// TIA Portal V19 export
FUNCTION_BLOCK "Motor"   // FB126, LAD
TITLE = MOTOR MANAGER / SIMPLE MOTOR MANAGER
// stored: Access Published, MemoryReserve 100, SetENOAutomatically false
   VAR_INPUT
      MotorCtrl : "MotorCtrl";
      ThermalProtection : Bool;   // Thermal protection (0 =OK)
      FdbkRunning : Bool;   // Contactor feedback
      FeedbackTimeout : Time := T#1S;   // Contatr feedback timeout
      Simulation : Bool;   // Simulation device
   END_VAR
   VAR_OUTPUT
      MotorSts : "MotorSts";
      Contactor : Bool;
   END_VAR
   VAR_IN_OUT
      Alarm : "MotorAlr";
   END_VAR
   VAR
      DelayContactorFeedbackON : IEC_TIMER;
      Ctrl_RunContactor : Bool;
   END_VAR
   VAR_TEMP
      DelayOnStart : Bool;
      DelayOffStart : Bool;
      AlarmPresence : Bool;
      RunPermitted : Bool;
   END_VAR
BEGIN

REGION Network 1 (SCL): Info
   //=============================================================================
   //PM FORMING
   //-----------------------------------------------------------------------------
   // Library: StandardBlocks
   // Tested with: S7-1518TF
   // Engineering: TIA Portal V18
   // Restrictions: -
   // Requirements: S7-1500
   // Functionality: Motor device manager
   //
   // v1.0.0  28/12/2022 
   // v1.1.0  23/01/2023 Added Simulation Input
   //=============================================================================
END_REGION

REGION Network 2: Alarm reset
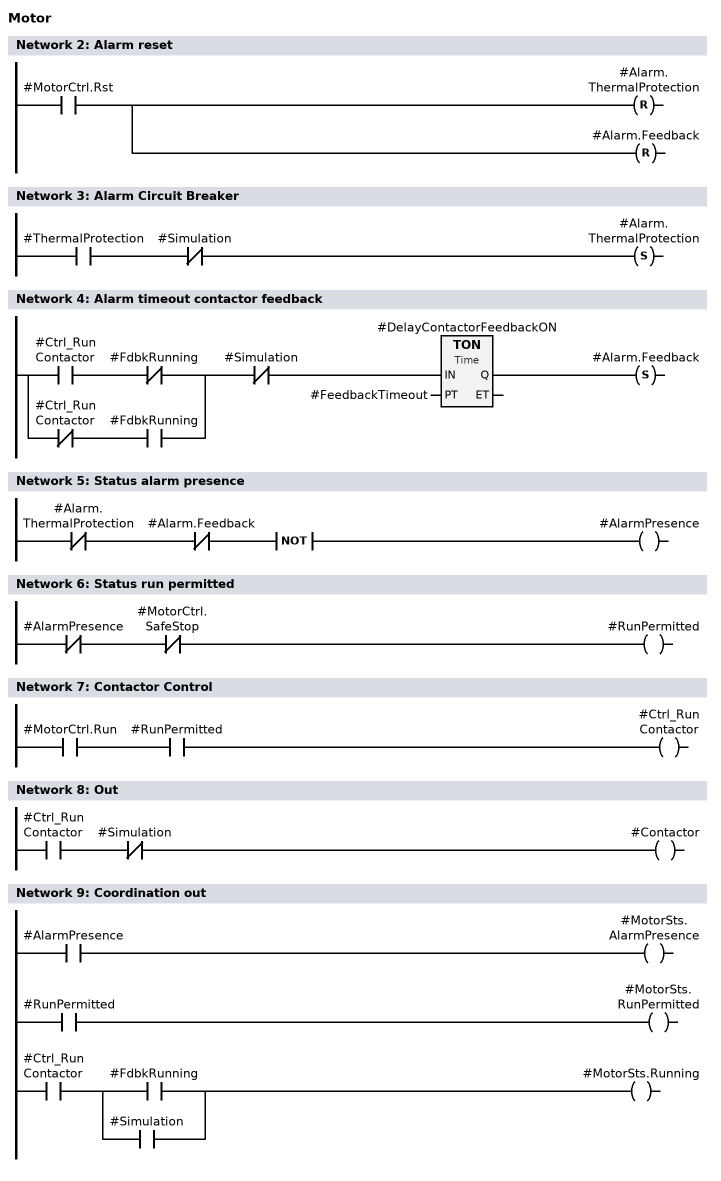
   RUNG wire#powerrail
      Contact( #MotorCtrl.Rst )
      wire#w1
      R_Coil( #Alarm.ThermalProtection )
   END_RUNG
   RUNG wire#w1
      R_Coil( #Alarm.Feedback )
   END_RUNG
   // the same network as SCL:
   IF #MotorCtrl.Rst THEN
       #Alarm.ThermalProtection := FALSE;
       #Alarm.Feedback := FALSE;
   END_IF;
END_REGION

REGION Network 3: Alarm Circuit Breaker
   RUNG wire#powerrail
      Contact( #ThermalProtection )
      I_Contact( #Simulation )
      S_Coil( #Alarm.ThermalProtection )
   END_RUNG
   // the same network as SCL:
   IF #ThermalProtection AND NOT #Simulation THEN #Alarm.ThermalProtection := TRUE; END_IF;
END_REGION

REGION Network 4: Alarm timeout contactor feedback
   RUNG wire#powerrail
      Contact( #Ctrl_RunContactor )
      I_Contact( #FdbkRunning )
      wire#w1
      I_Contact( #Simulation )
      { S7_Templates := "time_type := Time" } #DelayContactorFeedbackON.TON(pt := #FeedbackTimeout, et =>)
      S_Coil( #Alarm.Feedback )
   END_RUNG
   RUNG wire#powerrail
      I_Contact( #Ctrl_RunContactor )
      Contact( #FdbkRunning )
   END_RUNG wire#w1
   // the same network as SCL:
   #DelayContactorFeedbackON.TON(IN := ((#Ctrl_RunContactor AND NOT #FdbkRunning) OR (NOT #Ctrl_RunContactor AND #FdbkRunning)) AND NOT #Simulation,
                           PT := #FeedbackTimeout);
   IF #DelayContactorFeedbackON.Q THEN #Alarm.Feedback := TRUE; END_IF;
END_REGION

REGION Network 5: Status alarm presence
   RUNG wire#powerrail
      I_Contact( #Alarm.ThermalProtection )
      I_Contact( #Alarm.Feedback )
      Not()
      Coil( #AlarmPresence )
   END_RUNG
   // the same network as SCL:
   #AlarmPresence := NOT (NOT #Alarm.ThermalProtection AND NOT #Alarm.Feedback);
END_REGION

REGION Network 6: Status run permitted
   RUNG wire#powerrail
      I_Contact( #AlarmPresence )
      I_Contact( #MotorCtrl.SafeStop )
      Coil( #RunPermitted )
   END_RUNG
   // the same network as SCL:
   #RunPermitted := NOT #AlarmPresence AND NOT #MotorCtrl.SafeStop;
END_REGION

REGION Network 7: Contactor Control
   RUNG wire#powerrail
      Contact( #MotorCtrl.Run )
      Contact( #RunPermitted )
      Coil( #Ctrl_RunContactor )
   END_RUNG
   // the same network as SCL:
   #Ctrl_RunContactor := #MotorCtrl.Run AND #RunPermitted;
END_REGION

REGION Network 8: Out
   RUNG wire#powerrail
      Contact( #Ctrl_RunContactor )
      I_Contact( #Simulation )
      Coil( #Contactor )
   END_RUNG
   // the same network as SCL:
   #Contactor := #Ctrl_RunContactor AND NOT #Simulation;
END_REGION

REGION Network 9: Coordination out
   RUNG wire#powerrail
      Contact( #AlarmPresence )
      Coil( #MotorSts.AlarmPresence )
   END_RUNG
   RUNG wire#powerrail
      Contact( #RunPermitted )
      Coil( #MotorSts.RunPermitted )
   END_RUNG
   RUNG wire#powerrail
      Contact( #Ctrl_RunContactor )
      wire#w1
      Contact( #FdbkRunning )
      wire#w2
      Coil( #MotorSts.Running )
   END_RUNG
   RUNG wire#w1
      Contact( #Simulation )
   END_RUNG wire#w2
   // the same network as SCL:
   #MotorSts.AlarmPresence := #AlarmPresence;
   #MotorSts.RunPermitted := #RunPermitted;
   #MotorSts.Running := #Ctrl_RunContactor AND (#FdbkRunning OR #Simulation);
END_REGION
END_FUNCTION_BLOCK
